// Mitsubishi GX Works2 project: QUINTO EJERCICIO   PLC: FX2N/FX2NC

PROGRAM MAIN
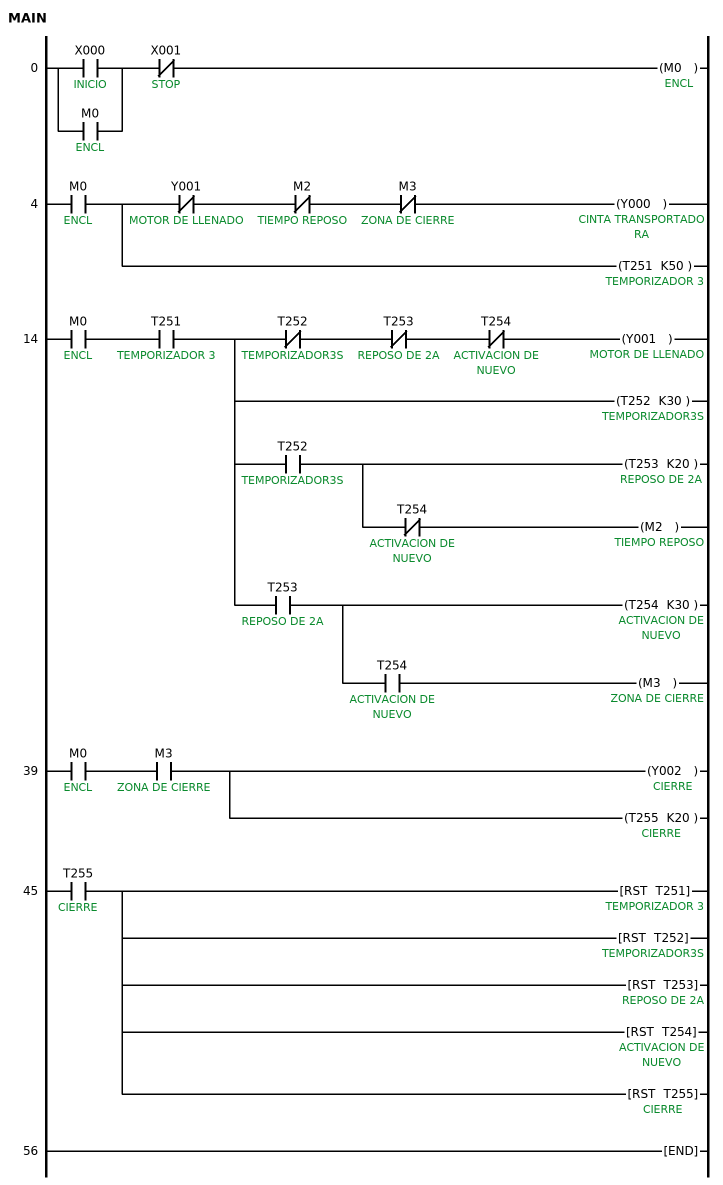
0     LD      X000  ; INICIO
      OR      M0  ; ENCL
      ANI     X001  ; STOP
      OUT     M0  ; ENCL
4     LD      M0  ; ENCL
      MPS
      ANI     Y001  ; MOTOR DE LLENADO
      ANI     M2  ; TIEMPO REPOSO
      ANI     M3  ; ZONA DE CIERRE
      OUT     Y000  ; CINTA TRANSPORTADORA
      MPP
      OUT     T251 K50  ; TEMPORIZADOR 3
14    LD      M0  ; ENCL
      AND     T251  ; TEMPORIZADOR 3
      MPS
      ANI     T252  ; TEMPORIZADOR3S
      ANI     T253  ; REPOSO DE 2A
      ANI     T254  ; ACTIVACION DE NUEVO
      OUT     Y001  ; MOTOR DE LLENADO
      MPP
      OUT     T252 K30  ; TEMPORIZADOR3S
      MPS
      AND     T252  ; TEMPORIZADOR3S
      OUT     T253 K20  ; REPOSO DE 2A
      ANI     T254  ; ACTIVACION DE NUEVO
      OUT     M2  ; TIEMPO REPOSO
      MPP
      AND     T253  ; REPOSO DE 2A
      OUT     T254 K30  ; ACTIVACION DE NUEVO
      AND     T254  ; ACTIVACION DE NUEVO
      OUT     M3  ; ZONA DE CIERRE
39    LD      M0  ; ENCL
      AND     M3  ; ZONA DE CIERRE
      OUT     Y002  ; CIERRE
      OUT     T255 K20  ; CIERRE
45    LD      T255  ; CIERRE
      RST     T251  ; TEMPORIZADOR 3
      RST     T252  ; TEMPORIZADOR3S
      RST     T253  ; REPOSO DE 2A
      RST     T254  ; ACTIVACION DE NUEVO
      RST     T255  ; CIERRE
56    END
END_PROGRAM

// device comments not shown above
T1  ; TEMPORIZADOR 1
T2  ; TEMPORIZADOR 3S
T3  ; REPOSO DE 2A
T4  ; ACTIVACION DE NUEVO
T5  ; CIERRE
T250  ; TEMPORIZADOR 1
